{attribute 'qualified_only'}
{attribute 'strict'}
TYPE ActivationStatus :
(
	Disabled,
	Enabled
);
END_TYPE

(* stored: Version 1.1.0.1, ProductVersion 3.1.4024.12
   DUT ActivationStatus: Id {e97029c7-f299-4ba4-a9e1-67f9bbdf7c4e} *)
